TEXTLIST TL_ConnectionState
  0 = 'Unknown'
  100 = 'Reset'
  101 = 'Session'
  102 = 'Connection'
  103 = 'Parameter'
  104 = 'Data'
  105 = 'Shutdown'
   = ''
END_TEXTLIST

(* stored: Version 1.1.0.1, ProductVersion 3.1.4022.12
   TextList TL_ConnectionState: Id {79679511-2869-4c23-8ffa-732b1bb97646} *)
